// TIA Portal V17 export
// export: Created 2022-01-04T17:38:23.1761518Z, ExportSetting WithDefaults, DisplayName Totally Integrated Automation Portal, DisplayVersion V17, DisplayName TIA Portal Openness, DisplayVersion V17, DisplayName TIA Portal Version Control Interface, DisplayVersion V17, DisplayName STEP 7 Professional, DisplayVersion V17, DisplayName STEP 7 Safety, DisplayVersion V17, DisplayName WinCC Advanced, DisplayVersion V17
DATA_BLOCK "IO"   // DB1
{ S7_Optimized_Access := 'TRUE' }
VERSION : 0.1
// stored: AutoNumber true, IsOnlyStoredInLoadMemory false, IsRetainMemResEnabled false, IsWriteProtectedInAS false, MemoryReserve 100
   VAR
      start : Bool;
      stop : Bool := true;
      awaryjeOproznianie : Bool := true;
      czasParzenia : Time := T#5S;
      zadanaIloscWody : Real := 500.0;
      zadanaIloscHerbaty : Real := 15.0;
      temperatura : Int;
      przenosnikM1 : Bool;
      mieszalnikM2 : Bool;
      podgrzewaczG1 : Bool;
      otworzZaworZ1 : Bool;
      otworzZasuweZ2 : Bool;
      otworzZasuweZ3 : Bool;
      wodaPoziom : Real;
      lisciePoziom : Real;
      glownyPoziom : Real;
   END_VAR
BEGIN
END_DATA_BLOCK
